{attribute 'qualified_only'}
{attribute 'strict'}
TYPE enum_CommandNumber :
(
	enum_member := 0
)DINT;
END_TYPE

(* stored: Version 1.1.0.1, ProductVersion 3.1.4024.4
   DUT enum_CommandNumber: Id {b59280a0-c718-4294-9529-6ff1b98251a6} *)
